{attribute 'no_explicit_call':= 'do not call this POU directly'}
FUNCTION_BLOCK TValueMonitor
VAR
    _CurrentValue : INT := -1;
    _PreviousValue : INT;
    _Changed : BOOL;
END_VAR

PROPERTY Changed : BOOL
GET
Changed := _Changed;
END_GET
END_PROPERTY

PROPERTY CurrentValue : INT
GET
CurrentValue := _CurrentValue;
END_GET
END_PROPERTY

PROPERTY PreviousValue : INT
GET
PreviousValue := _PreviousValue;
END_GET
END_PROPERTY

METHOD Reset
VAR_INPUT
END_VAR
_CurrentValue := 0;
_PreviousValue := 0;
END_METHOD

METHOD Test : BOOL
VAR_INPUT
    Value : INT;
END_VAR
_Changed := Value <> _CurrentValue;
_PreviousValue := _CurrentValue;
_CurrentValue := Value;

Test := _Changed;
END_METHOD

END_FUNCTION_BLOCK

(* stored: Version 1.1.0.1, ProductVersion 3.1.4024.3
   POU TValueMonitor: Id {591647b8-2c47-489b-b7d0-55ab105e2f90}, SpecialFunc None
   Property Changed: Id {be26849e-4211-41c6-a367-42df2289bdc3}
   Get Get: Id {0d633c53-6323-42ab-9a3d-584e47765771}
   Property CurrentValue: Id {d22ce7ec-c527-4370-9f47-f67132120b9e}
   Get Get: Id {d958010f-da6b-4a0d-a224-3e86cf8c8211}
   Property PreviousValue: Id {0f23966b-9af5-471f-8d31-07f21f96ea69}
   Get Get: Id {deb54991-94a8-4f18-af98-2b83cb9aa254}
   Method Reset: Id {dea024b2-1dee-467c-9832-1f68ebeca288}
   Method Test: Id {ecf9a3fe-9c14-44fa-ac8d-400c120ab469} *)
